(* Schneider Machine Expert - Basic project Programa_desafio02_gabarito, file version 2.7.0.0 *)
(* ProjectInformations: Name=Novo projeto *)

HARDWARE
  Cpu 0: TM221CE40T
  Cartridge1 0: TMC2AQ2V
  EthernetConfiguration: NetworkName=M221, IpAllocationMode=FixedAddress, IpAddress=10.200.4.104, SubnetMask=255.255.254.0
  EthernetConfiguration: NetworkName=M221, IpAllocationMode=FixedAddress, IpAddress=0.0.0.0, SubnetMask=0.0.0.0
  SerialLineConfiguration: Baud=Baud19200, Parity=ParityEven, DataBits=DataBits8, StopBits=StopBits1, PhysicalMedium=PhysicalMediumRs485, TransmissionMode=TransmissionModeModbusRtu, SlaveId=1, Addressing=SlaveAddressing
  MastTask: UsePeriodScanMode=false, PeriodScan=100
  FastTask: Period=255
  CpuBehavior: StartingMode=StartAsPreviousState, AutoSaveRamOnEeprom=true, WatchdogPeriod=250

SYMBOLS  (address, symbol, comment, settings)
  %M0       HABILITA
  %M1       INTERROMPE_ALARME
  %M2       ACIONAM_MANUAL
  %MW0      NIVEL
  %I0.8     BTN_LIGA
  %I0.9     BTN_DESLIGA
  %I0.10    EMERG
  %Q0.8     BOMBA
  %Q0.9     ALARME
  %IW0.0    SENSOR_NIVEL  [Type=Type_0_10V, Scope=Scope_Normal, Minimum=0, Maximum=1000]

POU Novo POU
  (* SectionNumber=1 *)

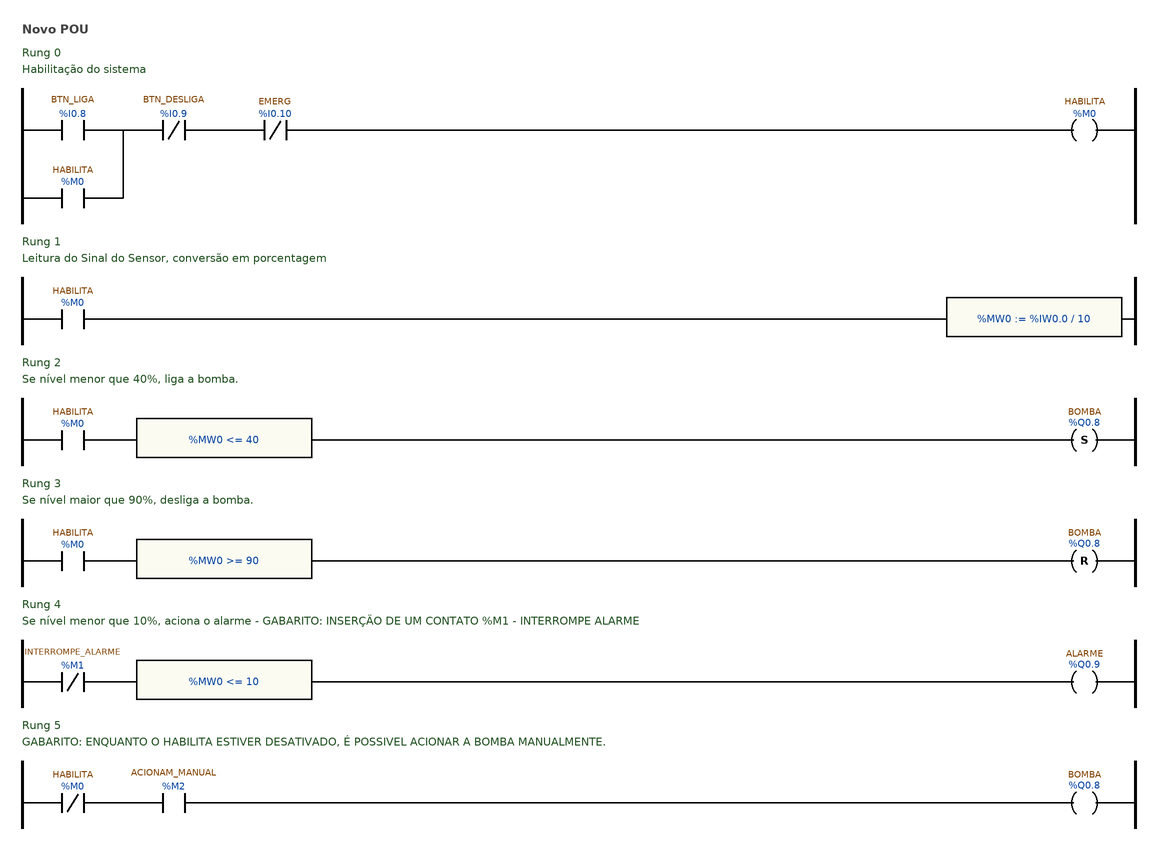

// Rung 0
// Habilitação do sistema
  LD %I0.8                (* BTN_LIGA *)
  OR %M0                  (* HABILITA *)
  ANDN %I0.9              (* BTN_DESLIGA *)
  ANDN %I0.10             (* EMERG *)
  ST %M0                  (* HABILITA *)
  // as ST:
  //   HABILITA := (BTN_LIGA OR HABILITA) AND NOT BTN_DESLIGA AND NOT EMERG;

// Rung 1
// Leitura do Sinal do Sensor, conversão em porcentagem
  LD %M0                  (* HABILITA *)
  [ %MW0 := %IW0.0 / 10 ] (* NIVEL, SENSOR_NIVEL *)
  // as ST:
  //   IF HABILITA THEN NIVEL := SENSOR_NIVEL / 10; END_IF;

// Rung 2
// Se nível menor que 40%, liga a bomba.
  LD %M0                  (* HABILITA *)
  AND [ %MW0 <= 40 ]      (* NIVEL *)
  S %Q0.8                 (* BOMBA *)
  // as ST:
  //   IF HABILITA AND NIVEL <= 40 THEN BOMBA := TRUE; END_IF;

// Rung 3
// Se nível maior que 90%, desliga a bomba.
  LD %M0                  (* HABILITA *)
  AND [ %MW0 >= 90 ]      (* NIVEL *)
  R %Q0.8                 (* BOMBA *)
  // as ST:
  //   IF HABILITA AND NIVEL >= 90 THEN BOMBA := FALSE; END_IF;

// Rung 4
// Se nível menor que 10%, aciona o alarme - GABARITO: INSERÇÃO DE UM CONTATO %M1 - INTERROMPE ALARME
  LDN %M1                 (* INTERROMPE_ALARME *)
  AND [ %MW0 <= 10 ]      (* NIVEL *)
  ST %Q0.9                (* ALARME *)
  // as ST:
  //   ALARME := NOT INTERROMPE_ALARME AND NIVEL <= 10;

// Rung 5
// GABARITO: ENQUANTO O HABILITA ESTIVER DESATIVADO, É POSSIVEL ACIONAR A BOMBA MANUALMENTE.
  LDN %M0                 (* HABILITA *)
  AND %M2                 (* ACIONAM_MANUAL *)
  ST %Q0.8                (* BOMBA *)
  // as ST:
  //   BOMBA := NOT HABILITA AND ACIONAM_MANUAL;
